FUNCTION_BLOCK FB_HE_SATT_FilterHolder IMPLEMENTS I_HE_SATT_FilterHolder
VAR
END_VAR


METHOD FB_Init: BOOL
VAR_INPUT
    bInitRetains: BOOL; // TRUE: the retain variables are initialized (reset warm / reset cold)
    bInCopyCode: BOOL;  // TRUE: the instance will be copied to the copy code afterward (online change)

//     iMotionStage : I_MotionStage;  
END_VAR
END_METHOD

{warning 'Add method implementation '}
METHOD GetFilter : I_HE_SATT_Filter
VAR_INPUT
	nFilterNumber	: INT;
END_VAR
END_METHOD


METHOD MoveToFilter
VAR_INPUT
    iFilter : I_HE_SATT_Filter;
    fThickness : LREAL;
END_VAR
END_METHOD

{warning 'Add property implementation'}
PROPERTY NumberOfSlots : INT
GET
END_GET
END_PROPERTY

{warning 'Add method implementation '}
METHOD RegisterFilter
VAR_INPUT
	iFilter	: I_HE_SATT_Filter;
END_VAR
END_METHOD

{warning 'Add property implementation'}
PROPERTY Status : REFERENCE TO ST_HE_SATT_Status
GET
END_GET
END_PROPERTY

END_FUNCTION_BLOCK

(* stored: Version 1.1.0.1
   POU FB_HE_SATT_FilterHolder: Id {b304d3c6-0dc8-4a7a-9624-8e9a7095a200}, SpecialFunc None
   Method FB_Init: Id {d3d486b6-acb1-4c10-9c60-66d79ba27f34}
   Method GetFilter: Id {dcf6eccc-ae4f-4d88-87a5-95aa1f4ace9d}
   Method MoveToFilter: Id {f0e6fc12-47bc-4b32-b594-9d75e111e828}
   Property NumberOfSlots: Id {51acaa5e-3c0e-4900-9c99-5692eeb6943b}
   Get Get: Id {f3e2489d-0230-4304-9a46-62762f15fd78}
   Method RegisterFilter: Id {278e3d4c-d878-46b2-bbd8-9700c44f35a5}
   Property Status: Id {93b2128b-bca4-43fd-a301-b4934c80cc9c}
   Get Get: Id {3bbfaabc-1721-498f-8a0f-1fc7ebd28d64} *)
